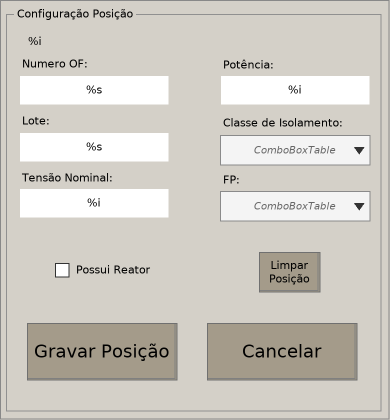
VISUALIZATION ConfigPosicao  // 390x420
VAR_IN_OUT
	bReator: BOOL;
	iOFnumber: INT;
	iSrlNumber: INT;
	
	
	
END_VAR
    GroupBox (6,6 375x405), "Configuração Posição"
        Checkbox (47,251 110x26), "Possui Reator", variable: gravarConfigPosicao.bReator[GVL.actEst]
        Button (21,317 150x57), "Gravar Posição"
            OnMouseClick: CloseDialog Dialog=ConfigPosicao, Result=OK, NumpadKeypadSet=True
            OnMouseClick: execute { gravarConfigPosicao(); }
        Button (201,317 150x57), "Cancelar"
            OnMouseClick: CloseDialog Dialog=ConfigPosicao, Result=Cancel, NumpadKeypadSet=True
        Button (253,246 61x40), "Limpar Posição"
            OnMouseClick: CloseDialog Dialog=ConfigPosicao, Result=Cancel, NumpadKeypadSet=True
            OnMouseClick: execute {
                gvl_p.aPositionsE019[gvl.actPos].numOF:='0';
                gvl_p.aPositionsE019[gvl.actPos].lote:='0';
                gvl_p.aPositionsE019[gvl.actPos].class:=0;
                gvl_p.aPositionsE019[gvl.actPos].pot:=0;
                gvl_p.aPositionsE019[gvl.actPos].cor:=0;
                IF gvl.totalPos[gvl.actEst] <> 0 THEN
                gvl.totalPos[gvl.actEst]:= gvl.totalPos[gvl.actEst] - 1;
                ELSE
                	gvl.totalPos[gvl.actEst] := 0;
                END_IF
                gravarConfigPosicao.bReator[0]:= false;
                ///// GERADOR DE LOG -------------------------------------------------------------
                gvl.envialog:= 'Posição Nº ';
                gvl.envialog:= concat(gvl.envialog, INT_TO_STRING(gvl.actPos));
                gvl.envialog:= concat(gvl.envialog,' foi limpa. ESTUFA 019');
                gvl.logRegister19:= gvl.envialog;
            }
        Label (13,43 81x30), "Numero OF:"
    Rectangle (24,30 22x23), "%i", text variable: GVL.actPos
    Textfield (19,75 150x30), "%s", text variable: GVL.cfgPos_OF019
        OnMouseDown: write the text variable via VisuDialogs.Numpad
    Label (19,163 111x30), "Tensão Nominal:"
    Textfield (220,75 150x30), "%i", text variable: GVL.cfgPos_Pot019
        OnMouseDown: write the text variable via VisuDialogs.Numpad
    Label (19,106 81x30), "Lote:"
    Label (220,165 56x30), "FP:"
    Label (220,108 144x30), "Classe de Isolamento:"
    Textfield (19,188 150x30), "%i", text variable: GVL.cfgPos_Class019
        OnMouseDown: write the text variable via VisuDialogs.Numpad
    Label (220,50 56x30), "Potência:"
    Textfield (19,132 150x30), "%s", text variable: GVL.cfgPos_LT019
        OnMouseDown: write the text variable via VisuDialogs.Keypad
    ComboBoxTable (220,135 150x30), variable: GVL.cfgPos_Iso019, data array: GVL_P.arr_Iso_1
        p3854506369: GVL_P.arr_Iso_1[INDEX]
    ComboBoxTable (220,191 150x30), variable: GVL.cfgPos_FP019, data array: GVL_P.arr_FP_1
        p3854506369: GVL_P.arr_FP_1[INDEX]
END_VISUALIZATION

(* stored: Version 1.1.0.1, ProductVersion 3.1.4024.12
   Visu ConfigPosicao: Id {a6174f95-717c-4e04-bf54-2d0ebd257176} *)
